INTERFACE I_LimSwStatusMCS2 EXTENDS I_LimSwStatus

PROPERTY InternalLimitActive : BOOL
GET
END_GET
SET
END_SET
END_PROPERTY

METHOD InternalLimits
VAR_INPUT
	InternalLimitActive : BOOL;
	WarningCondition : BOOL;
END_VAR
END_METHOD

PROPERTY LimOverride : BOOL
GET
END_GET
SET
END_SET
END_PROPERTY

PROPERTY MoveBackwardEnabled : BOOL
GET
END_GET
END_PROPERTY

PROPERTY MoveForwardEnabled : BOOL
GET
END_GET
END_PROPERTY

PROPERTY WarningCondition : BOOL
GET
END_GET
SET
END_SET
END_PROPERTY

END_INTERFACE

(* stored: Version 1.1.0.1
   Itf I_LimSwStatusMCS2: Id {7af97861-54c2-446c-8935-c4e0b207e519}
   Property InternalLimitActive: Id {aac82614-7e4e-4729-8fbe-2613d8825bf8}
   Get Get: Id {f2a06f00-b918-4808-96e8-1b2dd4a9ffef}
   Set Set: Id {b847d996-efbc-43e7-b79e-792df835eed5}
   Method InternalLimits: Id {35299885-28e2-415e-b733-185e9142885c}
   Property LimOverride: Id {c2b7a081-8622-4513-a352-40676732ddd4}
   Get Get: Id {92b682c9-0ed3-485f-b512-98fdd46e0b06}
   Set Set: Id {8cce1dba-985c-4025-a1be-c4f8cd661fe0}
   Property MoveBackwardEnabled: Id {de572613-9d45-4994-b1ca-1a9cc33027ab}
   Get Get: Id {fe29607c-fa72-4713-949d-b854b4bbd148}
   Property MoveForwardEnabled: Id {fb7daac9-08b3-40e8-ba2b-252151fa276c}
   Get Get: Id {f693efb7-a5a4-47bf-9045-f12740bf961e}
   Property WarningCondition: Id {b7bf2183-6b6f-4275-a585-bb63c58bc293}
   Get Get: Id {9ffd8b02-f22d-4839-9e05-58e7a2f50269}
   Set Set: Id {b7028200-0560-43f2-bf68-2d01168da6b8} *)
